(* PLC project CoDeSys External Library Template, WAGO e!COCKPIT e!COCKPIT, author 3S - Smart Software Solutions GmbH *)
(* stored: creationDateTime 2019-10-29T12:37:19.7040014, version 3.5.5.30, modificationDateTime 2019-10-29T12:36:39.3744516, organization 3S - Smart Software Solutions GmbH *)
(* Library project template with all possible element types, docu and a sample project structure *)

FUNCTION_BLOCK fbPPPSSilownikSABp
  VAR_INPUT
    sKomunikat : alSTRINGKomunikat;  (* komunikat z systemu zewnętrznego *)
    intTablicaKomunikatowRozmiar : INT;  (* rozmiar tablicy danych wysyłkowych *)
    intModbusOdczytZapisZadanieRozmiar : INT;  (* rozmiar tablicy danych modbusa *)
    xTablicaKomunikatowHold : BOOL;  (* wstrzymanie komunikacji mniej ważnych komunikatów *)
    sIdInstancji : STRING;  (* parametr ID rolety np NS02L*202IBM**** *)
    sIdAplikacji : STRING;  (* parametr ID aplikacji np SO*******ECL*000 *)
    sMnemonik : STRING;  (* mnemonik właściciela - BCB* *)
    sMACAdres : STRING;  (* MAC adres sterownika *)
    sDaneZapasowe : STRING;  (* 6 znaków zapasu *)
    tCzasOpoznieniaRestartu : TIME;  (* czas opóźnienia po którym zaczynają być raportowane wartości *)
    bAdres : BYTE;
    bKanalEnOcean : BYTE;
    sEnOceanID : STRING(10);
    rZadanePolozenieSilownika : REAL;
    tMinimalnyCzasRaportowania : TIME;
    tMaksymalnyCzasRaportowania : TIME;
    tCzasTimeoutEnOcean : TIME;
    xAutonomizacja : BOOL;
    xAutonomizacjaSztuczna : BOOL;
    xGlobalnaAutomatycznaKonfiguracja : BOOL;
    tCzestotliwoscAutomatycznejKonfiguracji : TIME;
    rTrybPracyAutonomizacja : REAL;  (* Domyślny tryb pracy *)
    rPozycjaSilownikaManAutonomizacja : REAL;  (* Domyślne położenie siłownika *)
    rFlagaSerwisowaAutonomizacja : REAL;  (* Domyślna flaga serwisowa *)
    tCzasSpadkuTemperatury : TIME;  (* Okres detekcji *)
    rDeltaSpadkuTemperatury : REAL;  (* Wartość o jaką musi spaść temp. w okresie intCzasSpadkuTemperatury, aby wyzwolić alarm *)
    rDeltaWzrostuTemperatury : REAL;  (* Wartość o jaką musi wzrosnąć temp. w okresie intCzasSpadkuTemperatury, aby odwołać alarm *)
    intTrybPracyHMI : INT := 1;  (* patrz enumPPPSZadajnikTrybPracy *)
    rZadanePolozenieSilownikaHMI : REAL;  (* Pozycja siłownika z nastawy na webvisu *)
    xPokazPanelHMI : BOOL := TRUE;  (* 0 - widoczny; 1 - niewidoczny *)
    xUsuwaniePotwierdzenieHMI : BOOL := FALSE;  (* wyświetlenie okienka potwierdzenia chęci usunięcia siłownika *)
    xUczenieWlaczHMI : BOOL := FALSE;  (* Włączenie flagi uczenia siłownika *)
    xUczenieWlaczone : BOOL;  (* Potwierdzenie włączenia uczenia *)
    xUsuwanieHMI : BOOL := FALSE;  (* Usuwanie EnOcean ID z kanału bramki *)
  END_VAR
  VAR_IN_OUT
    arModbusOdczytCykliczny : ARRAY[1..5000] OF typModbusOdczytCykliczny;
    arModbusStatusKomunikacji : ARRAY[1..256] OF INT;
    arModbusOdczytZapisZadanie : ARRAY[1..1000] OF typModbusOdczytZapisZadanie;
    intModbusOdczytZapisZadanieZnacznikZapisu : INT;
    arTablicaKomunikatow : alARRAYTablicaKomunikatow;
    intTablicaKomunikatowZnacznikZapisu : INT;
  END_VAR
  VAR_OUTPUT
    rDiagnostykaTemperaturaPomieszczenia : REAL;
    rDiagnostykaPozycjaSilownika : REAL;
    intDiagnostykaFlagaSerwisowa : INT;
    intDiagnostykaTrybPracy : INT;
    xDiagnostykaDetekcjaOtwarciaOkna : BOOL;
    sDiagnostykaEnOceanIDodczytany : STRING(10);
    xDiagnostykaPoprawneParowanie : BOOL;
    wDiagnostykaCzasOdOstatniegoKomunikatu : WORD;
  END_VAR
  VAR CONSTANT
    uintLiczbaRejestrowNaKanal : UINT := 20;
    uintPierwszyRejestr : UINT := 2000;
  END_VAR
  VAR
    wLearnEnOceanOdczytany : WORD;
    xLearnEnOceanOdczytany : BOOL;
    xLearnEnOceanWlacz : BOOL;
    xLearnEnOceanWylacz : BOOL;
    fbWysylanieLearn : TON;
    intTemp : INT := 0;
    xResetWysylanieLern : BOOL;
    xPoprawneParowanie : BOOL;
    uintORGModbusAdres : UINT;  (* definicja adresów rejestrów modbusowych *)
    uintFunctionModbusAdres : UINT;
    uintTypeModbusAdres : UINT;
    uintManufacturerModbusAdres : UINT;
    uintEnOceanIDHiModbusAdres : UINT;
    uintEnOceanIDLoModbusAdres : UINT;
    uintCzasOdOstatniegoKomunikatuModbusAdres : UINT;
    uintZadanaPozycjaSilownikaModbusAdres : UINT;
    uintFlagaSerwisowaModbusAdres : UINT;
    uintStatusUrzadzeniaModbusAdres : UINT;
    uintTemperaturaPomieszczeniaOdczytanaModbusAdres : UINT;
    uintNastawaPotencjometraModbusAdres : UINT;
    uintUczenieSilownikaAdres : UINT := 31;  (* uintLiczbaTelegramowModbusAdres : UINT; *)
    uintLearnModbusAdres : UINT;
    xPierwszySkan : BOOL := TRUE;  (* zmienne operacyjne *)
    intPetlaPierwszySkan : INT := 1;
    intRozkazTymczasowy : INT;
    rtrigPrzywrocDomyslne : R_TRIG;  (* Przywracanie domyślnych wartości nastaw *)
    rtrigZapisModbus : R_TRIG;  (* Triger zapisu danych po Modbusie *)
    fbTaktowanieZapisywaniaModbus : TON;  (* Cykliczne żądanie zapisu danych do urządzenia *)
    tonBrakKomunikacjiPLC : TON;  (* Kontrola komunikacji urządzenia *)
    xBrakKomunikacjiPLC : BOOL;
    xBrakKomunikacjiIZE : BOOL;
    fbWyslanieKonfiguracji : TON;  (* definicja zmiennych i FB do odczytu wartości z modbusa *)
    xPozwolenieNaAutomatycznaKonfiguracje : BOOL;
    xResetTimerautomatycznejKonfiguracji : BOOL;
    intBlokadaWykonywaniaRozkazow : INT;
    intBlokadaWykonywaniaRozkazowZaraportowana : INT;
    intTrybPracy : INT;  (* Tryb pracy regulatora. *)
    intTrybPracyPamiec : INT;
    intTrybPracyZaraportowana : INT;
    xTrybPracyZapisz : BOOL;  (* Trigger zapisu wartości w pamięci urządzenia. *)
    rTrybPracyZapis : REAL;  (* Wartość do zapisania w pamięci urządzenia. *)
    wFunctionEnOceanOdczytana : WORD;
    wTypeEnOceanOdczytana : WORD;
    wManufacturerEnOceanOdczytana : WORD;
    sEnOceanIDodczytany : STRING(10);
    wEnOceanIDHi : WORD;
    wEnOceanIDLo : WORD;
    wEnOceanIDHiZapis : WORD;
    wEnOceanIDLoZapis : WORD;
    wCzasOdOstatniegoKomunikatu : WORD;
    fbTimeoutEnOcean : TON;
    wStatusUrzadzenia : WORD;
    xBladBaterii : BOOL;
    fbBladBaterii : TON;
    xAlarmOgolny : BOOL;
    fbDecToBin : fbDecToBin;
    wLiczbaTelegramow : WORD;
    uintLiczbaTelegramow : UINT;
    wTemperaturaPomieszczeniaOdczytana : WORD;
    fbTemperaturaPomieszczenia : fbFiltrWartoscAnalogowa;
    rTemperaturaPomieszczenia : REAL := 273.15;
    rTemperaturaPomieszczeniaZaraportowana : REAL;
    rTemperaturaPomieszczeniaPamiec : REAL;  (* Temperatura zapamiętana w celu porównania z aktualną *)
    xBrakZmianyTemperatury : BOOL;  (* Flaga braku zmiany temperatury *)
    fbBrakZmianyTemperaturyTimer : TON;  (* Timer braku zmiany temperatury (24 godziny) *)
    xBladBrakZmianyTemperatury : BOOL;  (* Błąd braku zmiany temperatury *)
    wPozycjaSilownikaOdczytana : WORD;
    wPozycjaSilownikaZadanie : WORD;
    fbPozycjaSilownika : fbFiltrWartoscAnalogowa;
    rPozycjaSilownika : REAL;  (* Pozycja siłownika. *)
    rPozycjaSilownikaZaraportowana : REAL;
    rPozycjaSilownikaAuto : REAL;  (* Pozycja siłownika w trybie automatycznym. *)
    rPozycjaSilownikaAutoZaraportowana : REAL;
    rPozycjaSilownikaMan : REAL;  (* Pozycja siłownika w trybie manualnym *)
    rPozycjaSilownikaManZaraportowana : REAL;
    xPozycjaSilownikaManZapisz : BOOL;  (* Trigger zapisu wartości w pamięci urządzenia. *)
    rPozycjaSilownikaManZapis : REAL;  (* Wartość do zapisania w pamięci urządzenia. *)
    fbUtrzymaniaPolozeniaAutonomizacja : TON;
    xRestartTimeraUtrzymaniaPolozeniaAutonomizacja : BOOL;
    xWykonanoZapisPolozeniaSilownika : BOOL := FALSE;
    tCzasWyslaniaKomunikatuZapisuPozycjiSilownika : TIME;
    wFlagaSerwisowaOdczytana : WORD;
    wFlagaSerwisowaZadanie : WORD;
    intFlagaSerwisowa : INT;
    intFlagaSerwisowaZaraportowana : INT;
    xFlagaSerwisowaZapisz : BOOL;  (* Trigger zapisu wartości w pamięci urządzenia. *)
    rFlagaSerwisowaZapis : REAL;  (* Wartość do zapisania w pamięci urządzenia. *)
    xZmianaFlagiSerwisowejNaBrakDzialan : BOOL;
    xZmianaFlagiSerwisowejNaTrybLetni : BOOL;
    xZmianaFlagiSerwisowejNaZamkniecieZaworu : BOOL;
    xZmianaFlagiSerwisowejNaOtwarcieZaworu : BOOL;
    xZmianaFlagiSerwisowejNaPozycjaGorna : BOOL;
    xZmianaFlagiSerwisowejNaKalibracjeSilownika : BOOL;
    fbTimerZmianyFlagiSerwisowej : TON;
    xPoInicjalizacji : BOOL := FALSE;  (* inicjalizacja *)
    fbInicjalizacyjnyTimer : TON;
    sDane : alSTRINGKomunikat;
    sWyslanyKomunikat : alSTRINGKomunikat;
    sKomunikatPamiec : alSTRINGKomunikat;
    sWyslanyKomunikatDummy : alSTRINGKomunikat;
    intPetla : INT;
    arErrorStan : ARRAY[0..5] OF INT;  (* tablica przechowująca statusy alarmowe *)
    arErrorKlasa : ARRAY[0..5] OF INT;  (* tablica przechowująca klasy danych alarmów *)
    sTempWartoscAtrybutu : STRING;
    xRaport : BOOL;
    rNastawaPolozeniaSilownika : REAL;
    xAlarmOtwarciaOkna : BOOL;  (* Alarm detekcji gwałtownego spadku temperatury siłownika (otwarcia okna nad grzejnikiem) *)
    rTemperaturaPomieszczeniaHistoryczna : REAL;  (* Wartość temperatury zapisywana co intCzasSpadkuTemperatury w celu obliczenia różnicy *)
    fbDetekcjaOtwarciaOknaTimer : TON;  (* Timer detekcji otwarcia okna *)
    xDefrost : BOOL;  (* Defrost *)
    fbDefrostTimer : TON;
    rtrigDefrostTimer : R_TRIG;
    fbDefrostOdwolanie : TON;
    fnUczenieTimer : TON;  (* Timer uczenia *)
    fnWlaczenieUczenia : R_TRIG;  (* Włączenie uczenie na panelu HMI *)
    fnWylaczenieUczenia : F_TRIG;  (* Wyłączenie uczenia na panelu HMI *)
    fnUczenieZakonczone : F_TRIG;  (* Uczenie zostało zakończone *)
    xBrakKomunikacjiEnOcean : BOOL;  (* Brak komunikacji z urządzeniem po enOcean *)
    xAwariaUrzadzenia : BOOL;  (* Alarm ogólny *)
    rTempWartoscAtrybutu : REAL;
    intTempWartoscAtrybutu : INT;
    xDetekcjaOtwarciaOkna : BOOL;
  END_VAR

            (*			
Autor:					Paweł Kąkol, 2018-08-23-PK; Artur Wyszomirski; Jan Bartczak
Prawa majątkowe: 		Solwena Sp. z o.o., 
Aktualizacje:			
						2018-08-27-PK: dodanie algorytmu nadpisywania konfiguracji (uczenia) anteny
						2018-09-04-PK: dodanie rozkazu C, dodanie zapytań Q, dodanie raportowania M, dodanie alarmowania
						2018-09-10-PK: zmiana alarmowania braku komunikacji z Modbus RTU na alarmowanie timeout komunikacji EnOcean
						2018-09-12-PK: zaremowanie kodu uczącego bramkę, dodanie możliwości uczenia (LearnMode) ze zmiennej BOOL, sprawdzanie poprawności zainstalowania urządzenia (po EnOceanID)
						2018-09-25-AW: obsługa trybów manualnego i automatycznego
						2018-10-01-JB: dodanie ręcznej zmiany flagi serwisowej siłownika, zmiana sposobu zapisywania wartości wysterowania siłownika 
						2018-10-03-JB: poprawienie odczytywania kodów błędów
						2018-23-10-JB: przygotowanie atrybutów i alarmów do komunikacji z IZE
						2018-11-16-AW: inicjalizacja uczenia siłowników z programy
						2018-12-11-JB: zmiana sposobu działania alarmu z błędem baterii. Do momentu pierwszego odczytu wartości za pomocą ModbusRTU generowała się błędna informacja o błędzie baterii. 			
						2018-12-11-JB: skasowanie obsługi detekcji okna, ponieważ ten siłownik tego nie zawiera. 	
						2018-12-12-JB: napisanie od nowa obsługi ramek typu C i Q
						2019-01-04-AWy: detekcja otwarcia okna
						2019-01-28-JC: defrost
						2019-02-14-AWy: wysyłanie alarmu czujnika temperatury
						2019-02-27-JB: zmiana deadbandów w filtrach analogowych
						2019-03-20-AWy: uczenie siłownika z poziomu panelu HMI
						2019-03-21-AWy: usuwanie siłownika z poziomu panelu HMI
						2019-05-16-AWy: modyfikacja warunku na raportowanie. Dopisane: AND arModbusStatusKomunikacji[bAdres] = enumModbusStatus.KomunikacjaPrawidlowa AND xPoInicjalizacji 
						2019-05-20-AWy: - zmiana zachowania Defrostu. Po wykryciu spadku temperatury poniżej 8 stopni następuje przełączenie w tryb ręczny i odpalanie siłownika na 100%. 
										- alarm odwołany i powrót do normalnej pracy po osiągnięciu temperatury powyżej 10 stopni.
						2019-06-06-AWy: załadowanie domyślnych trybów pracy i nastaw po przejściu w tryb autonomizacji.
						2019-08-14-AWy: zmiana algorytmu defrostu ze względu na zmianę sposobu wybierania trybów pracy. Zmiana fbPrzywrocDomyslne z przerzutnika RS na R_TRIG.
						2019-09-17-AWy: usunięcie buga z defrostu.
						2019-09-23-AWy: modyfikacja generowania wartości zmiennej xBrakKomunikacjiPLC.
						2019-10-09-AWy: uzależnienie wystąpienia alarmu braku zmiany temperatury od stanu komunikacji.
						2019-10-18-AWy: dodanie atrybutu POZ.
						2019-10-22-AWy: - usunięcie uintLiczbaTelegramowModbusAdres z odczytu po Modbusie;
										- wydłużenie czasu fbTaktowanieZapisywaniaModbus oraz wprowadzenie trigera zapisu po Modbusie;
										- dodanie warunku poprawnej komunikacji przy generowaniu defrostu.
						2019-10-24-AWy: zmiana deadbandu fbPozycjaSilownika
												
Opis:					fb służy do komunikacji po Modbus RTU za pośrednictwem bramek (STC65-RS485) EnOcean z siłownikami HRU0 (SAB+) na budynkach PPP Sopot (ENGIE) 
*)

// Inicjalizacja sterownika
fbInicjalizacyjnyTimer(IN := NOT xPoInicjalizacji , PT := tCzasOpoznieniaRestartu);
IF fbInicjalizacyjnyTimer.Q THEN
	rTemperaturaPomieszczeniaZaraportowana := rTemperaturaPomieszczenia;
	rPozycjaSilownikaZaraportowana := rPozycjaSilownika;
	rPozycjaSilownikaAutoZaraportowana := rPozycjaSilownikaAuto;
	rPozycjaSilownikaManZaraportowana := rPozycjaSilownikaMan;
	intFlagaSerwisowaZaraportowana := intFlagaSerwisowa;
	xPoInicjalizacji := TRUE;
END_IF

// Włącz autonomizację jeśli sterownik jest w stanie inicjalizacji lub nastąpiło wymuszenie autonomizacji
IF NOT xPoInicjalizacji OR xAutonomizacjaSztuczna = TRUE THEN
	xAutonomizacja := TRUE;
END_IF 

// Kontrola komunikacji
tonBrakKomunikacjiPLC(IN := (wCzasOdOstatniegoKomunikatu > 180 OR arModbusStatusKomunikacji[bAdres] <> enumModbusStatus.KomunikacjaPrawidlowa), PT := T#180S);
IF tonBrakKomunikacjiPLC.Q THEN
	xBrakKomunikacjiPLC := TRUE;
ELSE
	xBrakKomunikacjiPLC := FALSE;
END_IF

IF xAutonomizacja THEN
	xBrakKomunikacjiIZE := TRUE;
ELSE
	xBrakKomunikacjiIZE := FALSE;
END_IF

// Deklaracja rejestrów Modbusa
IF xPierwszySkan THEN
	xPierwszySkan := FALSE;
	WHILE arModbusOdczytCykliczny[intPetlaPierwszySkan].bAdresUrzadzenia <> 0 DO
		intPetlaPierwszySkan := intPetlaPierwszySkan + 1;
	END_WHILE
	
	//wyznaczenie adresów rejestrów modbusowych
	uintORGModbusAdres := uintPierwszyRejestr + (uintLiczbaRejestrowNaKanal * (BYTE_TO_UINT(bKanalEnOcean) - 1));
	uintFunctionModbusAdres := uintORGModbusAdres + 1;
	uintTypeModbusAdres := uintORGModbusAdres + 2;
	uintManufacturerModbusAdres := uintORGModbusAdres + 3;
	uintEnOceanIDHiModbusAdres := uintORGModbusAdres + 4;
	uintEnOceanIDLoModbusAdres := uintORGModbusAdres + 5;
	uintCzasOdOstatniegoKomunikatuModbusAdres := uintORGModbusAdres + 6;
	uintZadanaPozycjaSilownikaModbusAdres := uintORGModbusAdres + 7;
	uintFlagaSerwisowaModbusAdres := uintORGModbusAdres + 8;
	uintStatusUrzadzeniaModbusAdres := uintORGModbusAdres + 9;
	uintTemperaturaPomieszczeniaOdczytanaModbusAdres := uintORGModbusAdres + 10;
	//uintLiczbaTelegramowModbusAdres := uintORGModbusAdres + 19;
	
	uintLearnModbusAdres := 31 + BYTE_TO_UINT(bKanalEnOcean);
	
//deklaracja rejestrow do odczytu
	//coil
	arModbusOdczytCykliczny[intPetlaPierwszySkan].bAdresUrzadzenia := bAdres;
	arModbusOdczytCykliczny[intPetlaPierwszySkan].bFunkcja := TO_BYTE(enumModbusKodyFunkcji.OdczytWyjscBitowych);
	arModbusOdczytCykliczny[intPetlaPierwszySkan].uiAdresRejestru := uintLearnModbusAdres;
	arModbusOdczytCykliczny[intPetlaPierwszySkan].ltCzestotliwosc := LTIME#1S;
	arModbusOdczytCykliczny[intPetlaPierwszySkan].pZmiennaReferencyjna := ADR(wLearnEnOceanOdczytany);
	intPetlaPierwszySkan := intPetlaPierwszySkan + 1;
	//rejestry
	arModbusOdczytCykliczny[intPetlaPierwszySkan].bAdresUrzadzenia := bAdres;
	arModbusOdczytCykliczny[intPetlaPierwszySkan].bFunkcja := TO_BYTE(enumModbusKodyFunkcji.OdczytNRejestrow);
	arModbusOdczytCykliczny[intPetlaPierwszySkan].uiAdresRejestru := uintFunctionModbusAdres;
	arModbusOdczytCykliczny[intPetlaPierwszySkan].ltCzestotliwosc := TIME_TO_LTIME(tMinimalnyCzasRaportowania);
	arModbusOdczytCykliczny[intPetlaPierwszySkan].pZmiennaReferencyjna := ADR(wFunctionEnOceanOdczytana);
	intPetlaPierwszySkan := intPetlaPierwszySkan + 1;
	
	arModbusOdczytCykliczny[intPetlaPierwszySkan].bAdresUrzadzenia := bAdres;
	arModbusOdczytCykliczny[intPetlaPierwszySkan].bFunkcja := TO_BYTE(enumModbusKodyFunkcji.OdczytNRejestrow);
	arModbusOdczytCykliczny[intPetlaPierwszySkan].uiAdresRejestru := uintTypeModbusAdres;
	arModbusOdczytCykliczny[intPetlaPierwszySkan].ltCzestotliwosc := TIME_TO_LTIME(tMinimalnyCzasRaportowania);
	arModbusOdczytCykliczny[intPetlaPierwszySkan].pZmiennaReferencyjna := ADR(wTypeEnOceanOdczytana);
	intPetlaPierwszySkan := intPetlaPierwszySkan + 1;
	
	arModbusOdczytCykliczny[intPetlaPierwszySkan].bAdresUrzadzenia := bAdres;
	arModbusOdczytCykliczny[intPetlaPierwszySkan].bFunkcja := TO_BYTE(enumModbusKodyFunkcji.OdczytNRejestrow);
	arModbusOdczytCykliczny[intPetlaPierwszySkan].uiAdresRejestru := uintManufacturerModbusAdres;
	arModbusOdczytCykliczny[intPetlaPierwszySkan].ltCzestotliwosc := TIME_TO_LTIME(tMinimalnyCzasRaportowania);
	arModbusOdczytCykliczny[intPetlaPierwszySkan].pZmiennaReferencyjna := ADR(wManufacturerEnOceanOdczytana);
	intPetlaPierwszySkan := intPetlaPierwszySkan + 1;
	
	arModbusOdczytCykliczny[intPetlaPierwszySkan].bAdresUrzadzenia := bAdres;
	arModbusOdczytCykliczny[intPetlaPierwszySkan].bFunkcja := TO_BYTE(enumModbusKodyFunkcji.OdczytNRejestrow);
	arModbusOdczytCykliczny[intPetlaPierwszySkan].uiAdresRejestru := uintEnOceanIDHiModbusAdres;
	arModbusOdczytCykliczny[intPetlaPierwszySkan].ltCzestotliwosc := TIME_TO_LTIME(tMinimalnyCzasRaportowania);
	arModbusOdczytCykliczny[intPetlaPierwszySkan].pZmiennaReferencyjna := ADR(wEnOceanIDHi);
	intPetlaPierwszySkan := intPetlaPierwszySkan + 1;
	
	arModbusOdczytCykliczny[intPetlaPierwszySkan].bAdresUrzadzenia := bAdres;
	arModbusOdczytCykliczny[intPetlaPierwszySkan].bFunkcja := TO_BYTE(enumModbusKodyFunkcji.OdczytNRejestrow);
	arModbusOdczytCykliczny[intPetlaPierwszySkan].uiAdresRejestru := uintEnOceanIDLoModbusAdres;
	arModbusOdczytCykliczny[intPetlaPierwszySkan].ltCzestotliwosc := TIME_TO_LTIME(tMinimalnyCzasRaportowania);
	arModbusOdczytCykliczny[intPetlaPierwszySkan].pZmiennaReferencyjna := ADR(wEnOceanIDLo);
	intPetlaPierwszySkan := intPetlaPierwszySkan + 1;
	
	arModbusOdczytCykliczny[intPetlaPierwszySkan].bAdresUrzadzenia := bAdres;
	arModbusOdczytCykliczny[intPetlaPierwszySkan].bFunkcja := TO_BYTE(enumModbusKodyFunkcji.OdczytNRejestrow);
	arModbusOdczytCykliczny[intPetlaPierwszySkan].uiAdresRejestru := uintCzasOdOstatniegoKomunikatuModbusAdres;
	arModbusOdczytCykliczny[intPetlaPierwszySkan].ltCzestotliwosc := TIME_TO_LTIME(tMinimalnyCzasRaportowania);
	arModbusOdczytCykliczny[intPetlaPierwszySkan].pZmiennaReferencyjna := ADR(wCzasOdOstatniegoKomunikatu);
	intPetlaPierwszySkan := intPetlaPierwszySkan + 1;
	
	arModbusOdczytCykliczny[intPetlaPierwszySkan].bAdresUrzadzenia := bAdres;
	arModbusOdczytCykliczny[intPetlaPierwszySkan].bFunkcja := TO_BYTE(enumModbusKodyFunkcji.OdczytNRejestrow);
	arModbusOdczytCykliczny[intPetlaPierwszySkan].uiAdresRejestru := uintZadanaPozycjaSilownikaModbusAdres;
	arModbusOdczytCykliczny[intPetlaPierwszySkan].ltCzestotliwosc := TIME_TO_LTIME(tMinimalnyCzasRaportowania);
	arModbusOdczytCykliczny[intPetlaPierwszySkan].pZmiennaReferencyjna := ADR(wPozycjaSilownikaOdczytana);
	intPetlaPierwszySkan := intPetlaPierwszySkan + 1;	
	
	arModbusOdczytCykliczny[intPetlaPierwszySkan].bAdresUrzadzenia := bAdres;
	arModbusOdczytCykliczny[intPetlaPierwszySkan].bFunkcja := TO_BYTE(enumModbusKodyFunkcji.OdczytNRejestrow);
	arModbusOdczytCykliczny[intPetlaPierwszySkan].uiAdresRejestru := uintFlagaSerwisowaModbusAdres;
	arModbusOdczytCykliczny[intPetlaPierwszySkan].ltCzestotliwosc := TIME_TO_LTIME(tMinimalnyCzasRaportowania);
	arModbusOdczytCykliczny[intPetlaPierwszySkan].pZmiennaReferencyjna := ADR(wFlagaSerwisowaOdczytana);
	intPetlaPierwszySkan := intPetlaPierwszySkan + 1;
	
	arModbusOdczytCykliczny[intPetlaPierwszySkan].bAdresUrzadzenia := bAdres;
	arModbusOdczytCykliczny[intPetlaPierwszySkan].bFunkcja := TO_BYTE(enumModbusKodyFunkcji.OdczytNRejestrow);
	arModbusOdczytCykliczny[intPetlaPierwszySkan].uiAdresRejestru := uintStatusUrzadzeniaModbusAdres;
	arModbusOdczytCykliczny[intPetlaPierwszySkan].ltCzestotliwosc := TIME_TO_LTIME(tMinimalnyCzasRaportowania);
	arModbusOdczytCykliczny[intPetlaPierwszySkan].pZmiennaReferencyjna := ADR(wStatusUrzadzenia);
	intPetlaPierwszySkan := intPetlaPierwszySkan + 1;
	
	arModbusOdczytCykliczny[intPetlaPierwszySkan].bAdresUrzadzenia := bAdres;
	arModbusOdczytCykliczny[intPetlaPierwszySkan].bFunkcja := TO_BYTE(enumModbusKodyFunkcji.OdczytNRejestrow);
	arModbusOdczytCykliczny[intPetlaPierwszySkan].uiAdresRejestru := uintTemperaturaPomieszczeniaOdczytanaModbusAdres;
	arModbusOdczytCykliczny[intPetlaPierwszySkan].ltCzestotliwosc := TIME_TO_LTIME(tMinimalnyCzasRaportowania);
	arModbusOdczytCykliczny[intPetlaPierwszySkan].pZmiennaReferencyjna := ADR(wTemperaturaPomieszczeniaOdczytana);
	intPetlaPierwszySkan := intPetlaPierwszySkan + 1;
(*	
	arModbusOdczytCykliczny[intPetlaPierwszySkan].bAdresUrzadzenia := bAdres;
	arModbusOdczytCykliczny[intPetlaPierwszySkan].bFunkcja := TO_BYTE(enumModbusKodyFunkcji.OdczytNRejestrow);
	arModbusOdczytCykliczny[intPetlaPierwszySkan].uiAdresRejestru := uintLiczbaTelegramowModbusAdres;
	arModbusOdczytCykliczny[intPetlaPierwszySkan].ltCzestotliwosc := TIME_TO_LTIME(tMinimalnyCzasRaportowania);
	arModbusOdczytCykliczny[intPetlaPierwszySkan].pZmiennaReferencyjna := ADR(wLiczbaTelegramow);
	intPetlaPierwszySkan := intPetlaPierwszySkan + 1;
*)			
	arModbusOdczytCykliczny[intPetlaPierwszySkan].bAdresUrzadzenia := bAdres;
	arModbusOdczytCykliczny[intPetlaPierwszySkan].bFunkcja := TO_BYTE(enumModbusKodyFunkcji.OdczytWyjscBitowych);
	arModbusOdczytCykliczny[intPetlaPierwszySkan].uiAdresRejestru := uintUczenieSilownikaAdres + BYTE_TO_UINT(bKanalEnOcean);
	arModbusOdczytCykliczny[intPetlaPierwszySkan].ltCzestotliwosc := TIME_TO_LTIME(tMinimalnyCzasRaportowania);
	arModbusOdczytCykliczny[intPetlaPierwszySkan].pZmiennaReferencyjna := ADR(xUczenieWlaczone);
	intPetlaPierwszySkan := intPetlaPierwszySkan + 1;
END_IF

//obsluga komunikatu przychodzacego z IZE

IF 	sKomunikat <> sKomunikatPamiec AND xPoInicjalizacji THEN
	sKomunikatPamiec := sKomunikat;
	IF fnIDOdbiorcyMatch(sKomunikat , sIdInstancji) THEN
		sDane := '';
		//rozkaz typu C
		IF fnKomunikatTyp(sKomunikat) = 'C' AND NOT xAutonomizacja THEN
		//blokada
			IF fnKomunikatDaneSzukajWartosci(sKomunikat,'BLOK=') = '0' THEN
				IF intBlokadaWykonywaniaRozkazow = 1 THEN
					intBlokadaWykonywaniaRozkazow := 0;
					xRaport := TRUE;
					ELSE	
					IF sDane <> '' THEN
					sDane := CONCAT(sDane , ';');
					END_IF
					sDane := CONCAT(sDane , 'BLOK=0');
				END_IF
			END_IF
			IF fnKomunikatDaneSzukajWartosci(sKomunikat,'BLOK=') = '1' THEN
				IF intBlokadaWykonywaniaRozkazow = 0 THEN
					intBlokadaWykonywaniaRozkazow := 1;
					xRaport := TRUE;
					ELSE
					IF sDane <> '' THEN
					sDane := CONCAT(sDane , ';');
					END_IF					
					sDane := CONCAT(sDane , 'BLOK=1');
				END_IF
			END_IF
			
			IF intBlokadaWykonywaniaRozkazow = 0 THEN
				// Tryby pracy 
				fnKomunikatDaneZnajdzPorownajZapisz(sKomunikat := sKomunikat,
					sAtrybut := 'TRYB=',
					rAtrybutWartosc := rTrybPracyZapis,
					sDane := sDane,
					xAtrybutZapisz => xTrybPracyZapisz);		
				// Pozycja siłownika w trybie manualnym
				fnKomunikatDaneZnajdzPorownajZapisz(sKomunikat := sKomunikat,
					sAtrybut := 'POZMAN=',
					rAtrybutWartosc := rPozycjaSilownikaManZapis,
					sDane := sDane,
					xAtrybutZapisz => xPozycjaSilownikaManZapisz);
				// Flaga serwisowa
				fnKomunikatDaneZnajdzPorownajZapisz(sKomunikat := sKomunikat,
					sAtrybut := 'SERWIS=',
					rAtrybutWartosc := rFlagaSerwisowaZapis,
					sDane := sDane,
					xAtrybutZapisz => xFlagaSerwisowaZapisz);	
			END_IF	
		END_IF		

		//zapytanie typu Q
		IF fnKomunikatTyp(sKomunikat) = 'Q' AND arModbusStatusKomunikacji[bAdres] = enumModbusStatus.KomunikacjaPrawidlowa THEN
			IF fnKomunikatDaneSzukajWartosci(sKomunikat , 'BLOK=') = '?' OR fnKomunikatDaneSzukajWartosci(sKomunikat , 'ALL=') = '?' THEN
				fnKomunikatDaneDodaj(sDane := sDane , sAtrybut := 'BLOK=' , sWartosc := INT_TO_STRING(intBlokadaWykonywaniaRozkazow));	
			END_IF
			IF fnKomunikatDaneSzukajWartosci(sKomunikat , 'TRYB=') = '?' OR fnKomunikatDaneSzukajWartosci(sKomunikat , 'ALL=') = '?' THEN
				fnKomunikatDaneDodaj(sDane := sDane , sAtrybut := 'TRYB=' , sWartosc := INT_TO_STRING(intTrybPracy));	
			END_IF
			IF fnKomunikatDaneSzukajWartosci(sKomunikat , 'TEMP=') = '?' OR fnKomunikatDaneSzukajWartosci(sKomunikat , 'ALL=') = '?' THEN
				fnKomunikatDaneDodaj(sDane := sDane , sAtrybut := 'TEMP=' , sWartosc := REAL_TO_STRING(rTemperaturaPomieszczenia));	
			END_IF
			IF fnKomunikatDaneSzukajWartosci(sKomunikat , 'POZ=') = '?' OR fnKomunikatDaneSzukajWartosci(sKomunikat , 'ALL=') = '?' THEN
				fnKomunikatDaneDodaj(sDane := sDane , sAtrybut := 'POZ=' , sWartosc := REAL_TO_STRING(rPozycjaSilownika));	
			END_IF
			IF fnKomunikatDaneSzukajWartosci(sKomunikat , 'POZAUTO=') = '?' OR fnKomunikatDaneSzukajWartosci(sKomunikat , 'ALL=') = '?' THEN
				fnKomunikatDaneDodaj(sDane := sDane , sAtrybut := 'POZAUTO=' , sWartosc := REAL_TO_STRING(rPozycjaSilownikaAuto));	
			END_IF
			IF fnKomunikatDaneSzukajWartosci(sKomunikat , 'POZMAN=') = '?' OR fnKomunikatDaneSzukajWartosci(sKomunikat , 'ALL=') = '?' THEN
				fnKomunikatDaneDodaj(sDane := sDane , sAtrybut := 'POZMAN=' , sWartosc := REAL_TO_STRING(rPozycjaSilownikaMan / 100));	
			END_IF
			IF fnKomunikatDaneSzukajWartosci(sKomunikat , 'SERWIS=') = '?' OR fnKomunikatDaneSzukajWartosci(sKomunikat , 'ALL=') = '?' THEN
				fnKomunikatDaneDodaj(sDane := sDane , sAtrybut := 'SERWIS=' , sWartosc := INT_TO_STRING(intFlagaSerwisowa));	
			END_IF
			//pytanie o stany alarmów
			IF fnKomunikatDaneSzukajWartosci(sKomunikat , 'ALARM=') = '?' OR fnKomunikatDaneSzukajWartosci(sKomunikat , 'ALL=') = '?' THEN
				FOR intPetla := 1 TO 5 BY 1 DO
					//raportowanie typu E (stanów alarmów) na zapytanie typu Q
					IF arErrorStan[intPetla] <> enumAlarmWartosc.StanNieznany THEN
						fnZapiszKomunikat(	sCalyKomunikat := '' ,
											sTypKomunikatu := 'E' ,
											sMnemonik := sMnemonik ,
											sMACAdres := sMACAdres ,
											sIDNadawcy := sIdInstancji ,
											sIDOdbiorcy := sIdAplikacji ,
											sDaneZapasowe := sDaneZapasowe ,
											sDane := fnKomunikatDaneErrorRetry(xAktywny := arErrorStan[intPetla] = enumAlarmWartosc.StanAlarmowy , intKlasa := arErrorKlasa[intPetla] , intNumer := intPetla),
											arTablicaKomunikatow := arTablicaKomunikatow ,
											intTablicaKomunikatowZnacznikZapisu := intTablicaKomunikatowZnacznikZapisu ,
											intTablicaKomunikatowRozmiar := intTablicaKomunikatowRozmiar ,
											sWyslanyKomunikat := sWyslanyKomunikatDummy);
					END_IF
				END_FOR
			END_IF
		END_IF
		//raportowanie typu A
		IF sDane <> '' THEN
			fnZapiszKomunikat(	sCalyKomunikat := '' ,
								sTypKomunikatu := 'A' ,
								sMnemonik := sMnemonik ,
								sMACAdres := sMACAdres ,
								sIDNadawcy := sIdInstancji ,
								sIDOdbiorcy := sIdAplikacji ,
								sDaneZapasowe := sDaneZapasowe ,
								sDane := sDane ,
								arTablicaKomunikatow := arTablicaKomunikatow ,
								intTablicaKomunikatowZnacznikZapisu := intTablicaKomunikatowZnacznikZapisu ,
								intTablicaKomunikatowRozmiar := intTablicaKomunikatowRozmiar ,
								sWyslanyKomunikat := sWyslanyKomunikatDummy);
		END_IF
	END_IF
END_IF

// Przywrócenie wartości domyślnych nastaw krzywej grzewczej i trybów pracy w przypadku restartu sterownika lub przejścia w stan autonomizacji (brak komunikacji z IZE)
rtrigPrzywrocDomyslne(CLK := xAutonomizacja);
IF rtrigPrzywrocDomyslne.Q THEN	
	IF intTrybPracy <> REAL_TO_INT(rTrybPracyAutonomizacja) THEN
		rTrybPracyZapis := rTrybPracyAutonomizacja;
		xTrybPracyZapisz := TRUE;
	END_IF
	IF rPozycjaSilownikaMan <> rPozycjaSilownikaManAutonomizacja THEN
		rPozycjaSilownikaManZapis := rPozycjaSilownikaManAutonomizacja / 100;
		xPozycjaSilownikaManZapisz := TRUE;
	END_IF
	IF intFlagaSerwisowa <> REAL_TO_INT(rFlagaSerwisowaAutonomizacja) THEN
		rFlagaSerwisowaZapis :=  rFlagaSerwisowaAutonomizacja;
		xFlagaSerwisowaZapisz := TRUE;
	END_IF
END_IF	

// Zapisanie nastaw domyślnych lub otrzymanych w ramce C
IF xTrybPracyZapisz THEN
	intTrybPracy := REAL_TO_INT(rTrybPracyZapis);
	intTrybPracyHMI := REAL_TO_INT(rTrybPracyZapis);
	xTrybPracyZapisz := FALSE;
END_IF	
IF xPozycjaSilownikaManZapisz THEN
	rPozycjaSilownikaMan := rPozycjaSilownikaManZapis * 100;
	xPozycjaSilownikaManZapisz := FALSE;
END_IF	

// Trigger zapisu po Modbusie
rtrigZapisModbus (CLK := xFlagaSerwisowaZapisz);

// Taktowanie zapisywania po Modbusie
fbTaktowanieZapisywaniaModbus(IN := NOT fbTaktowanieZapisywaniaModbus.Q, PT := T#180S);
				
// Zapisywanie trybu pracy do pamięci urządzenia
IF xFlagaSerwisowaZapisz AND (fbTaktowanieZapisywaniaModbus.Q OR rtrigZapisModbus.Q) THEN
	fnModbusZapisRejestru(	bAdresUrzadzenia := bAdres,
							bFunkcja := INT_TO_BYTE(enumModbusKodyFunkcji.ZapisRejestru),
							uiAdresRejestru := uintFlagaSerwisowaModbusAdres,
							pZmiennaReferencyjna := 0,
							wWartoscDoZapisania := REAL_TO_WORD(rFlagaSerwisowaZapis),
							intModbusOdczytZapisZadanieRozmiar := intModbusOdczytZapisZadanieRozmiar,
							arModbusOdczytZapisZadanie := arModbusOdczytZapisZadanie,
							intModbusOdczytZapisZadanieZnacznikZapisu := intModbusOdczytZapisZadanieZnacznikZapisu);
	IF intFlagaSerwisowa = REAL_TO_INT(rFlagaSerwisowaZapis) THEN					
		xFlagaSerwisowaZapisz := FALSE;
	END_IF
END_IF

//Auto konfiguracja anteny - sprawdzenie czy EnOcean ID wpisany w EiG jest zgodny z tym odczytanym z kanalu bramki
sEnOceanIDodczytany := CONCAT(CONCAT(fnKonwersjaDEC_BYTE_TO_HEX_STRING(INT_TO_BYTE(WORD_TO_INT(wEnOceanIDHi / 256))), fnKonwersjaDEC_BYTE_TO_HEX_STRING(WORD_TO_BYTE(wEnOceanIDHi))), CONCAT(fnKonwersjaDEC_BYTE_TO_HEX_STRING(INT_TO_BYTE(WORD_TO_INT(wEnOceanIDLo / 256))), fnKonwersjaDEC_BYTE_TO_HEX_STRING(WORD_TO_BYTE(wEnOceanIDLo))));
IF sEnOceanIDodczytany = sEnOceanID THEN
	xPoprawneParowanie := TRUE;
ELSE
	xPoprawneParowanie := FALSE;
END_IF

//sprawdzanie Timeout komunikacji
fbTimeoutEnOcean(IN := ((wCzasOdOstatniegoKomunikatu > 180 OR wCzasOdOstatniegoKomunikatu = 0) AND arModbusStatusKomunikacji[bAdres] = enumModbusStatus.KomunikacjaPrawidlowa) , PT := tCzasTimeoutEnOcean);

// dokonywanie obliczeń
fbTemperaturaPomieszczenia(	rWartoscWejsciowa := WORD_TO_REAL(wTemperaturaPomieszczeniaOdczytana),
							rWartoscWejsciowaZaraportowana := rTemperaturaPomieszczeniaZaraportowana,
							rDeadband := 0.1,
							tCzasMinimalny := tMinimalnyCzasRaportowania,
							tCzasMaksymalny := tMaksymalnyCzasRaportowania,
							rWynikMnoznik := 0.1,
							rWynikOffset := 273.15,
							rWartoscWyjsciowa => rTemperaturaPomieszczenia);
							
fbPozycjaSilownika(			rWartoscWejsciowa := WORD_TO_REAL(wPozycjaSilownikaOdczytana),
							rWartoscWejsciowaZaraportowana := rPozycjaSilownikaZaraportowana,
							rDeadband := 0.1,
							tCzasMinimalny := tMinimalnyCzasRaportowania,
							tCzasMaksymalny := tMaksymalnyCzasRaportowania,
							rWynikMnoznik := 0.01,
							rWynikOffset := 0.0,
							rWartoscWyjsciowa => rPozycjaSilownika);
							
CASE WORD_TO_INT(wFlagaSerwisowaOdczytana) OF
	0 : intFlagaSerwisowa := enumPPPSSilownikSABpServiceFlag.BrakDzialan;
	9 : intFlagaSerwisowa := enumPPPSSilownikSABpServiceFlag.TrybLetni;
	17 : intFlagaSerwisowa := enumPPPSSilownikSABpServiceFlag.ZamkniecieZaworu;
	33 : intFlagaSerwisowa := enumPPPSSilownikSABpServiceFlag.OtwarcieZaworu;
	65 : intFlagaSerwisowa := enumPPPSSilownikSABpServiceFlag.PozycjaGorna;
	129 : intFlagaSerwisowa := enumPPPSSilownikSABpServiceFlag.KalibracjaSilownika;
END_CASE
	
fbDecToBin(	wWordWejsciowy := wStatusUrzadzenia, 
			intIloscBitow := 8);
												
xAlarmOgolny := BYTE_TO_BOOL(fbDecToBin.arBity[0]);

// Defrost silownika. 
// Po spadku temperatury siłownika poniżej 8 stopni siłownik jest ustawiany w pozycję pełnego otwarcia (w trybie manualnym). Po wzroście temperatury powyżej 10 stopni siłownik powraca do trybu automatycznego.
fbDefrostTimer(IN := (rTemperaturaPomieszczenia < 281.15) AND (arModbusStatusKomunikacji[bAdres] = enumModbusStatus.KomunikacjaPrawidlowa), PT := T#5M);	// Temperatura poniżej 8 stopni C przez okres 5 minut
rtrigDefrostTimer(CLK := fbDefrostTimer.Q);
IF rtrigDefrostTimer.Q THEN
	intTrybPracyPamiec := intTrybPracy;	
END_IF

IF fbDefrostTimer.Q THEN	// Ustaw tryb pracy na manualny i otwórz zawór na 100%. Uruchom alarm
	rTrybPracyZapis := enumPPPSSilownikTrybPracy.Manualny;
	xTrybPracyZapisz := TRUE;
	rPozycjaSilownikaManZapis := 1;
	xPozycjaSilownikaManZapisz := TRUE;
	rZadanePolozenieSilownikaHMI := 100;
	xDefrost := TRUE;	
END_IF

fbDefrostOdwolanie(IN := ((rTemperaturaPomieszczenia > 283.15) AND xDefrost), PT := T#5M);	// Temperatura powyżej 10 stopni i uruchomiony Defrost przez okres 5 minut
IF fbDefrostOdwolanie.Q THEN	// Ustawa tryb pracy na automatyczny i odwołaj alarm
	rTrybPracyZapis := intTrybPracyPamiec;
	xTrybPracyZapisz := TRUE;
	xDefrost := FALSE;
END_IF
//
											
// Tryby pracy 
IF xAutonomizacja THEN	
	IF intTrybPracyHMI = enumPPPSSilownikTrybPracy.Manualny THEN								// tryb ręczny na HMI
		intTrybPracy := enumPPPSSilownikTrybPracy.Manualny;	
		rNastawaPolozeniaSilownika := rZadanePolozenieSilownikaHMI;
		rPozycjaSilownikaMan := rNastawaPolozeniaSilownika;
	ELSE																						// tryb automatyczny HMI
		intTrybPracy := enumPPPSSilownikTrybPracy.Automatyczny;	
		rNastawaPolozeniaSilownika := rZadanePolozenieSilownika;
		rZadanePolozenieSilownikaHMI := rZadanePolozenieSilownika;	
		rPozycjaSilownikaAuto := rPozycjaSilownika;											
	END_IF
ELSE
	rZadanePolozenieSilownikaHMI := rNastawaPolozeniaSilownika;
	IF intTrybPracy = enumPPPSSilownikTrybPracy.Manualny THEN
		rNastawaPolozeniaSilownika := rPozycjaSilownikaMan;
		intTrybPracyHMI := enumPPPSZadajnikTrybPracy.Manualny;
	ELSE
		rNastawaPolozeniaSilownika := rZadanePolozenieSilownika;
		intTrybPracyHMI := enumPPPSZadajnikTrybPracy.Automatyczny;
		rPozycjaSilownikaAuto := rPozycjaSilownika;		
	END_IF
END_IF
		
//utrzymanie położenia
fbUtrzymaniaPolozeniaAutonomizacja(IN := xRestartTimeraUtrzymaniaPolozeniaAutonomizacja = TRUE, PT := tCzasWyslaniaKomunikatuZapisuPozycjiSilownika);

IF (INT_TO_WORD(REAL_TO_INT(rNastawaPolozeniaSilownika)) <> wPozycjaSilownikaOdczytana) THEN
		xRestartTimeraUtrzymaniaPolozeniaAutonomizacja := TRUE;
		IF xWykonanoZapisPolozeniaSilownika = FALSE THEN
			tCzasWyslaniaKomunikatuZapisuPozycjiSilownika := T#5s;	
		END_IF	
ELSE
	xRestartTimeraUtrzymaniaPolozeniaAutonomizacja := FALSE;	
	xWykonanoZapisPolozeniaSilownika := FALSE;
END_IF

IF fbUtrzymaniaPolozeniaAutonomizacja.Q AND arModbusStatusKomunikacji[bAdres] = enumModbusStatus.KomunikacjaPrawidlowa THEN
	fnModbusZapisRejestru(	bAdresUrzadzenia := bAdres,
							bFunkcja := INT_TO_BYTE(enumModbusKodyFunkcji.ZapisRejestru),
							uiAdresRejestru := uintZadanaPozycjaSilownikaModbusAdres,
							pZmiennaReferencyjna := 0,
							wWartoscDoZapisania := (INT_TO_WORD(REAL_TO_INT(rNastawaPolozeniaSilownika))),
							intModbusOdczytZapisZadanieRozmiar := intModbusOdczytZapisZadanieRozmiar,
							arModbusOdczytZapisZadanie := arModbusOdczytZapisZadanie,
							intModbusOdczytZapisZadanieZnacznikZapisu := intModbusOdczytZapisZadanieZnacznikZapisu);
	xRestartTimeraUtrzymaniaPolozeniaAutonomizacja := FALSE;
	tCzasWyslaniaKomunikatuZapisuPozycjiSilownika := T#45s;
	xWykonanoZapisPolozeniaSilownika := TRUE;
END_IF

// Uczenie siłownika do bramki
fnWlaczenieUczenia(CLK := xUczenieWlaczHMI);
fnWylaczenieUczenia(CLK := xUczenieWlaczHMI);
fnUczenieZakonczone(CLK := xUczenieWlaczone);

IF fnUczenieZakonczone.Q OR fnUczenieTimer.Q THEN																		// Jeśli FALSE na coilu uczenia opuść toggla na HMI
	xUczenieWlaczHMI := FALSE;		
END_IF

IF fnWlaczenieUczenia.Q THEN						
	fnModbusZapisRejestru(	bAdresUrzadzenia := bAdres,																	// Wystawienie TRUE na coilu uczenia (patrz dok. STC65 rozdział 2.5.2)
							bFunkcja := INT_TO_BYTE(enumModbusKodyFunkcji.ZapisBitu),
							uiAdresRejestru := 31 + BYTE_TO_UINT(bKanalEnOcean),
							pZmiennaReferencyjna := 0,
							wWartoscDoZapisania := (BOOL_TO_WORD(TRUE)),
							intModbusOdczytZapisZadanieRozmiar := intModbusOdczytZapisZadanieRozmiar,
							arModbusOdczytZapisZadanie := arModbusOdczytZapisZadanie,
							intModbusOdczytZapisZadanieZnacznikZapisu := intModbusOdczytZapisZadanieZnacznikZapisu);	
END_IF

fnUczenieTimer(IN := xUczenieWlaczone, PT := T#1M);																		// Czas na uczenie - 1 minuta 

IF fnWylaczenieUczenia.Q THEN
	fnModbusZapisRejestru(	bAdresUrzadzenia := bAdres,																	// Wystawienie FALSE na coilu uczenia (patrz dok. STC65 rozdział 2.5.2)
							bFunkcja := INT_TO_BYTE(enumModbusKodyFunkcji.ZapisBitu),
							uiAdresRejestru := 31 + BYTE_TO_UINT(bKanalEnOcean),
							pZmiennaReferencyjna := 0,
							wWartoscDoZapisania := (BOOL_TO_WORD(FALSE)),
							intModbusOdczytZapisZadanieRozmiar := intModbusOdczytZapisZadanieRozmiar,
							arModbusOdczytZapisZadanie := arModbusOdczytZapisZadanie,
							intModbusOdczytZapisZadanieZnacznikZapisu := intModbusOdczytZapisZadanieZnacznikZapisu);			
END_IF	
//

// Usuwanie siłownika z bramki
IF xUsuwanieHMI THEN	// Usuwanie EnOceanID z bramki
	fnModbusZapisRejestru(	bAdresUrzadzenia := bAdres,																	
							bFunkcja := INT_TO_BYTE(enumModbusKodyFunkcji.ZapisNRejestrow),
							uiAdresRejestru := uintEnOceanIDHiModbusAdres,
							pZmiennaReferencyjna := ADR(wEnOceanIDHi),
							wWartoscDoZapisania := 0,
							intModbusOdczytZapisZadanieRozmiar := intModbusOdczytZapisZadanieRozmiar,
							arModbusOdczytZapisZadanie := arModbusOdczytZapisZadanie,
							intModbusOdczytZapisZadanieZnacznikZapisu := intModbusOdczytZapisZadanieZnacznikZapisu);	
	fnModbusZapisRejestru(	bAdresUrzadzenia := bAdres,																	
							bFunkcja := INT_TO_BYTE(enumModbusKodyFunkcji.ZapisNRejestrow),
							uiAdresRejestru := uintEnOceanIDLoModbusAdres,
							pZmiennaReferencyjna := ADR(wEnOceanIDLo),
							wWartoscDoZapisania := 0,
							intModbusOdczytZapisZadanieRozmiar := intModbusOdczytZapisZadanieRozmiar,
							arModbusOdczytZapisZadanie := arModbusOdczytZapisZadanie,
							intModbusOdczytZapisZadanieZnacznikZapisu := intModbusOdczytZapisZadanieZnacznikZapisu);	
	xUsuwanieHMI := FALSE;					
END_IF
//
(*
// Zmiana koloru - po kliknięciu w symbol siłownika na HMI togglowana jest zmienna xZmienKolorHMI. xResetKoloruHMI resetuje kolor na symbolu, który był kliknięty wcześniej
IF xResetKoloruHMI THEN
	xKolorHMI := FALSE;
	xZmienKolorHMI := FALSE;
END_IF

IF xZmienKolorHMI THEN
	xKolorHMI := TRUE;
END_IF
//
*)
// Detekcja otwarcia okna (jeśli temperatura spadnie w czasie intCzasSpadkuTemperatury o rDeltaSpadkuTemperatury wystaw alarm. Zdejmij alarm, jeśli temp. wzrośnie o rDeltaWzrostuTemperatury
fbDetekcjaOtwarciaOknaTimer(IN := NOT(fbDetekcjaOtwarciaOknaTimer.Q), PT := tCzasSpadkuTemperatury);
IF fbDetekcjaOtwarciaOknaTimer.Q THEN
	rTemperaturaPomieszczeniaHistoryczna := rTemperaturaPomieszczenia;
END_IF
IF (rTemperaturaPomieszczeniaHistoryczna - rTemperaturaPomieszczenia) > rDeltaSpadkuTemperatury THEN
	xAlarmOtwarciaOkna := TRUE;
END_IF
IF (rTemperaturaPomieszczenia - rTemperaturaPomieszczeniaHistoryczna) > rDeltaWzrostuTemperatury THEN
	xAlarmOtwarciaOkna := FALSE;
END_IF
//
// Sprawdzanie czy pomiar temperatury działa (odczyt jest niepoprawny, jeśli nie zmienił wartości w przeciągu doby)
IF rTemperaturaPomieszczeniaPamiec = rTemperaturaPomieszczenia THEN
	xBrakZmianyTemperatury := TRUE;
ELSE
	xBrakZmianyTemperatury := FALSE;	
END_IF
fbBrakZmianyTemperaturyTimer(IN := xBrakZmianyTemperatury, PT := T#12H);
rTemperaturaPomieszczeniaPamiec := rTemperaturaPomieszczenia;
IF fbBrakZmianyTemperaturyTimer.Q AND NOT xBrakKomunikacjiPLC THEN
	xBladBrakZmianyTemperatury := TRUE;
ELSE
	xBladBrakZmianyTemperatury := FALSE;
END_IF
//
///////Diagnostyka na czas uruchomień////////
	rDiagnostykaTemperaturaPomieszczenia := rTemperaturaPomieszczenia;
	rDiagnostykaPozycjaSilownika := rPozycjaSilownika;
	intDiagnostykaFlagaSerwisowa := intFlagaSerwisowa;
	intDiagnostykaTrybPracy := intTrybPracy;
	sDiagnostykaEnOceanIDodczytany := sEnOceanIDodczytany;
	xDiagnostykaPoprawneParowanie := xPoprawneParowanie;
	wDiagnostykaCzasOdOstatniegoKomunikatu := wCzasOdOstatniegoKomunikatu;
//////////////////////////////////////////////				
							
					
//raportowanie		
IF (intBlokadaWykonywaniaRozkazow <> intBlokadaWykonywaniaRozkazowZaraportowana OR intTrybPracy <> intTrybPracyZaraportowana OR rTemperaturaPomieszczenia <> rTemperaturaPomieszczeniaZaraportowana OR 
	rPozycjaSilownika <> rPozycjaSilownikaZaraportowana OR intFlagaSerwisowa <> intFlagaSerwisowaZaraportowana OR rPozycjaSilownikaMan <> rPozycjaSilownikaManZaraportowana OR 
	rPozycjaSilownikaAuto <> rPozycjaSilownikaAutoZaraportowana) AND arModbusStatusKomunikacji[bAdres] = enumModbusStatus.KomunikacjaPrawidlowa AND xPoInicjalizacji THEN
	xRaport := TRUE;
END_IF

IF xRaport THEN
	sDane := '';
	xRaport := FALSE;
	IF intBlokadaWykonywaniaRozkazow <> intBlokadaWykonywaniaRozkazowZaraportowana THEN
		intBlokadaWykonywaniaRozkazowZaraportowana := intBlokadaWykonywaniaRozkazow;
		fnKomunikatDaneDodaj(sDane := sDane , sAtrybut := 'BLOK=' , sWartosc := INT_TO_STRING(intBlokadaWykonywaniaRozkazow));	
	END_IF
	IF intTrybPracy <> intTrybPracyZaraportowana THEN
		intTrybPracyZaraportowana := intTrybPracy;
		fnKomunikatDaneDodaj(sDane := sDane , sAtrybut := 'TRYB=' , sWartosc := INT_TO_STRING(intTrybPracy));	
	END_IF
	IF rTemperaturaPomieszczenia <> rTemperaturaPomieszczeniaZaraportowana THEN
		rTemperaturaPomieszczeniaZaraportowana := rTemperaturaPomieszczenia;
		fnKomunikatDaneDodaj(sDane := sDane , sAtrybut := 'TEMP=' , sWartosc := REAL_TO_STRING(rTemperaturaPomieszczenia));	
	END_IF
	IF rPozycjaSilownika <> rPozycjaSilownikaZaraportowana THEN
		rPozycjaSilownikaZaraportowana := rPozycjaSilownika;
		fnKomunikatDaneDodaj(sDane := sDane , sAtrybut := 'POZ=' , sWartosc := REAL_TO_STRING(rPozycjaSilownika));	
	END_IF
	IF rPozycjaSilownikaMan <> rPozycjaSilownikaManZaraportowana THEN
		rPozycjaSilownikaManZaraportowana := rPozycjaSilownikaMan;
		fnKomunikatDaneDodaj(sDane := sDane , sAtrybut := 'POZMAN=' , sWartosc := REAL_TO_STRING(rPozycjaSilownikaMan / 100));	
	END_IF
	IF rPozycjaSilownikaAuto <> rPozycjaSilownikaAutoZaraportowana THEN
		rPozycjaSilownikaAutoZaraportowana := rPozycjaSilownikaAuto;
		fnKomunikatDaneDodaj(sDane := sDane , sAtrybut := 'POZAUTO=' , sWartosc := REAL_TO_STRING(rPozycjaSilownikaAuto));	
	END_IF
	IF intFlagaSerwisowa <> intFlagaSerwisowaZaraportowana THEN
		intFlagaSerwisowaZaraportowana := intFlagaSerwisowa;
		fnKomunikatDaneDodaj(sDane := sDane , sAtrybut := 'SERWIS=' , sWartosc := INT_TO_STRING(intFlagaSerwisowa));	
	END_IF

	IF sDane <> '' AND xPoInicjalizacji THEN
		fnZapiszKomunikat(	sCalyKomunikat := '' ,
							sTypKomunikatu := 'M' ,
							sMnemonik := sMnemonik ,
							sMACAdres := sMACAdres ,
							sIDNadawcy := sIdInstancji ,
							sIDOdbiorcy := sIdAplikacji ,
							sDaneZapasowe := sDaneZapasowe ,
							sDane := sDane ,
							arTablicaKomunikatow := arTablicaKomunikatow ,
							intTablicaKomunikatowZnacznikZapisu := intTablicaKomunikatowZnacznikZapisu ,
							intTablicaKomunikatowRozmiar := intTablicaKomunikatowRozmiar ,
							sWyslanyKomunikat := sWyslanyKomunikat);
	END_IF
END_IF

// obsługa alarmów do siłownika
	//brak komunikacji po EnOcean
IF arErrorStan[enumPPPSSilownikSABpError.BrakKomunikacji] <> enumAlarmWartosc.StanAlarmowy AND fbTimeoutEnOcean.Q AND arModbusStatusKomunikacji[bAdres] = enumModbusStatus.KomunikacjaPrawidlowa THEN
	arErrorStan[enumPPPSSilownikSABpError.BrakKomunikacji] := enumAlarmWartosc.StanAlarmowy;
	xBrakKomunikacjiEnOcean := TRUE;
	arErrorKlasa[enumPPPSSilownikSABpError.BrakKomunikacji] := enumPPPSSilownikSABpErrorKlasa.BrakKomunikacji;
	IF xPoInicjalizacji THEN
		fnZapiszKomunikat(	sCalyKomunikat := '' ,
							sTypKomunikatu := 'E' ,
							sMnemonik := sMnemonik ,
							sMACAdres := sMACAdres ,
							sIDNadawcy := sIdInstancji ,
							sIDOdbiorcy := sIdAplikacji ,
							sDaneZapasowe := sDaneZapasowe ,
							sDane := fnKomunikatDaneError(xAktywny := TRUE , intKlasa := enumPPPSSilownikSABpErrorKlasa.BrakKomunikacji , intNumer := enumPPPSSilownikSABpError.BrakKomunikacji),
							arTablicaKomunikatow := arTablicaKomunikatow ,
							intTablicaKomunikatowZnacznikZapisu := intTablicaKomunikatowZnacznikZapisu ,
							intTablicaKomunikatowRozmiar := intTablicaKomunikatowRozmiar ,
							sWyslanyKomunikat := sWyslanyKomunikatDummy);
	END_IF
END_IF
IF arErrorStan[enumPPPSSilownikSABpError.BrakKomunikacji] <> enumAlarmWartosc.StanNormalny AND NOT fbTimeoutEnOcean.Q AND arModbusStatusKomunikacji[bAdres] = enumModbusStatus.KomunikacjaPrawidlowa THEN
	arErrorStan[enumPPPSSilownikSABpError.BrakKomunikacji] := enumAlarmWartosc.StanNormalny;
	xBrakKomunikacjiEnOcean := FALSE;
	arErrorKlasa[enumPPPSSilownikSABpError.BrakKomunikacji] := enumPPPSSilownikSABpErrorKlasa.BrakKomunikacji;
	IF xPoInicjalizacji THEN
		fnZapiszKomunikat(	sCalyKomunikat := '' ,
							sTypKomunikatu := 'E' ,
							sMnemonik := sMnemonik ,
							sMACAdres := sMACAdres ,
							sIDNadawcy := sIdInstancji ,
							sIDOdbiorcy := sIdAplikacji ,
							sDaneZapasowe := sDaneZapasowe ,
							sDane := fnKomunikatDaneError(xAktywny := FALSE , intKlasa := enumPPPSSilownikSABpErrorKlasa.BrakKomunikacji , intNumer := enumPPPSSilownikSABpError.BrakKomunikacji),
							arTablicaKomunikatow := arTablicaKomunikatow ,
							intTablicaKomunikatowZnacznikZapisu := intTablicaKomunikatowZnacznikZapisu ,
							intTablicaKomunikatowRozmiar := intTablicaKomunikatowRozmiar ,
							sWyslanyKomunikat := sWyslanyKomunikatDummy);
	END_IF
END_IF
	//Alarm ogólny
IF arErrorStan[enumPPPSSilownikSABpError.AlarmOgolny] <> enumAlarmWartosc.StanAlarmowy AND xAlarmOgolny AND arModbusStatusKomunikacji[bAdres] = enumModbusStatus.KomunikacjaPrawidlowa THEN
	arErrorStan[enumPPPSSilownikSABpError.AlarmOgolny] := enumAlarmWartosc.StanAlarmowy;
	xAwariaUrzadzenia := TRUE;
	arErrorKlasa[enumPPPSSilownikSABpError.AlarmOgolny] := enumPPPSSilownikSABpErrorKlasa.AlarmOgolny;
	IF xPoInicjalizacji THEN
		fnZapiszKomunikat(	sCalyKomunikat := '' ,
							sTypKomunikatu := 'E' ,
							sMnemonik := sMnemonik ,
							sMACAdres := sMACAdres ,
							sIDNadawcy := sIdInstancji ,
							sIDOdbiorcy := sIdAplikacji ,
							sDaneZapasowe := sDaneZapasowe ,
							sDane := fnKomunikatDaneError(xAktywny := TRUE , intKlasa := enumPPPSSilownikSABpErrorKlasa.AlarmOgolny , intNumer := enumPPPSSilownikSABpError.AlarmOgolny),
							arTablicaKomunikatow := arTablicaKomunikatow ,
							intTablicaKomunikatowZnacznikZapisu := intTablicaKomunikatowZnacznikZapisu ,
							intTablicaKomunikatowRozmiar := intTablicaKomunikatowRozmiar ,
							sWyslanyKomunikat := sWyslanyKomunikatDummy);
	END_IF
END_IF
IF arErrorStan[enumPPPSSilownikSABpError.AlarmOgolny] <> enumAlarmWartosc.StanNormalny AND NOT xAlarmOgolny AND arModbusStatusKomunikacji[bAdres] = enumModbusStatus.KomunikacjaPrawidlowa THEN
	arErrorStan[enumPPPSSilownikSABpError.AlarmOgolny] := enumAlarmWartosc.StanNormalny;
	xAwariaUrzadzenia := FALSE;
	arErrorKlasa[enumPPPSSilownikSABpError.AlarmOgolny] := enumPPPSSilownikSABpErrorKlasa.AlarmOgolny;
	IF xPoInicjalizacji THEN
		fnZapiszKomunikat(	sCalyKomunikat := '' ,
							sTypKomunikatu := 'E' ,
							sMnemonik := sMnemonik ,
							sMACAdres := sMACAdres ,
							sIDNadawcy := sIdInstancji ,
							sIDOdbiorcy := sIdAplikacji ,
							sDaneZapasowe := sDaneZapasowe ,
							sDane := fnKomunikatDaneError(xAktywny := FALSE , intKlasa := enumPPPSSilownikSABpErrorKlasa.AlarmOgolny , intNumer := enumPPPSSilownikSABpError.AlarmOgolny),
							arTablicaKomunikatow := arTablicaKomunikatow ,
							intTablicaKomunikatowZnacznikZapisu := intTablicaKomunikatowZnacznikZapisu ,
							intTablicaKomunikatowRozmiar := intTablicaKomunikatowRozmiar ,
							sWyslanyKomunikat := sWyslanyKomunikatDummy);
	END_IF
END_IF
	// Detekcja otwarcia okna
IF arErrorStan[enumPPPSSilownikSABpError.DetekcjaOtwarciaOkna] <> enumAlarmWartosc.StanAlarmowy AND xDetekcjaOtwarciaOkna AND arModbusStatusKomunikacji[bAdres] = enumModbusStatus.KomunikacjaPrawidlowa THEN
	arErrorStan[enumPPPSSilownikSABpError.DetekcjaOtwarciaOkna] := enumAlarmWartosc.StanAlarmowy;
	arErrorKlasa[enumPPPSSilownikSABpError.DetekcjaOtwarciaOkna] := enumPPPSSilownikSABpErrorKlasa.DetekcjaOtwarciaOkna;
	IF xPoInicjalizacji THEN
		fnZapiszKomunikat(	sCalyKomunikat := '' ,
							sTypKomunikatu := 'E' ,
							sMnemonik := sMnemonik ,
							sMACAdres := sMACAdres ,
							sIDNadawcy := sIdInstancji ,
							sIDOdbiorcy := sIdAplikacji ,
							sDaneZapasowe := sDaneZapasowe ,
							sDane := fnKomunikatDaneError(xAktywny := TRUE , intKlasa := enumPPPSSilownikSABpErrorKlasa.DetekcjaOtwarciaOkna , intNumer := enumPPPSSilownikSABpError.DetekcjaOtwarciaOkna),
							arTablicaKomunikatow := arTablicaKomunikatow ,
							intTablicaKomunikatowZnacznikZapisu := intTablicaKomunikatowZnacznikZapisu ,
							intTablicaKomunikatowRozmiar := intTablicaKomunikatowRozmiar ,
							sWyslanyKomunikat := sWyslanyKomunikatDummy);
	END_IF
END_IF
IF arErrorStan[enumPPPSSilownikSABpError.DetekcjaOtwarciaOkna] <> enumAlarmWartosc.StanNormalny AND NOT xDetekcjaOtwarciaOkna AND arModbusStatusKomunikacji[bAdres] = enumModbusStatus.KomunikacjaPrawidlowa THEN
	arErrorStan[enumPPPSSilownikSABpError.DetekcjaOtwarciaOkna] := enumAlarmWartosc.StanNormalny;
	arErrorKlasa[enumPPPSSilownikSABpError.DetekcjaOtwarciaOkna] := enumPPPSSilownikSABpErrorKlasa.DetekcjaOtwarciaOkna;
	IF xPoInicjalizacji THEN
		fnZapiszKomunikat(	sCalyKomunikat := '' ,
							sTypKomunikatu := 'E' ,
							sMnemonik := sMnemonik ,
							sMACAdres := sMACAdres ,
							sIDNadawcy := sIdInstancji ,
							sIDOdbiorcy := sIdAplikacji ,
							sDaneZapasowe := sDaneZapasowe ,
							sDane := fnKomunikatDaneError(xAktywny := FALSE , intKlasa := enumPPPSSilownikSABpErrorKlasa.DetekcjaOtwarciaOkna , intNumer := enumPPPSSilownikSABpError.DetekcjaOtwarciaOkna),
							arTablicaKomunikatow := arTablicaKomunikatow ,
							intTablicaKomunikatowZnacznikZapisu := intTablicaKomunikatowZnacznikZapisu ,
							intTablicaKomunikatowRozmiar := intTablicaKomunikatowRozmiar ,
							sWyslanyKomunikat := sWyslanyKomunikatDummy);
	END_IF
END_IF
// Defrost
IF arErrorStan[enumPPPSSilownikSABpError.Defrost] <> enumAlarmWartosc.StanAlarmowy AND xDefrost AND arModbusStatusKomunikacji[bAdres] = enumModbusStatus.KomunikacjaPrawidlowa THEN
	arErrorStan[enumPPPSSilownikSABpError.Defrost] := enumAlarmWartosc.StanAlarmowy;
	arErrorKlasa[enumPPPSSilownikSABpError.Defrost] := enumPPPSSilownikSABpErrorKlasa.Defrost;
	IF xPoInicjalizacji THEN
		fnZapiszKomunikat(	sCalyKomunikat := '' ,
							sTypKomunikatu := 'E' ,
							sMnemonik := sMnemonik ,
							sMACAdres := sMACAdres ,
							sIDNadawcy := sIdInstancji ,
							sIDOdbiorcy := sIdAplikacji ,
							sDaneZapasowe := sDaneZapasowe ,
							sDane := fnKomunikatDaneError(xAktywny := TRUE , intKlasa := enumPPPSSilownikSABpErrorKlasa.Defrost , intNumer := enumPPPSSilownikSABpError.Defrost),
							arTablicaKomunikatow := arTablicaKomunikatow ,
							intTablicaKomunikatowZnacznikZapisu := intTablicaKomunikatowZnacznikZapisu ,
							intTablicaKomunikatowRozmiar := intTablicaKomunikatowRozmiar ,
							sWyslanyKomunikat := sWyslanyKomunikatDummy);
	END_IF
END_IF
IF arErrorStan[enumPPPSSilownikSABpError.Defrost] <> enumAlarmWartosc.StanNormalny AND NOT xDefrost AND arModbusStatusKomunikacji[bAdres] = enumModbusStatus.KomunikacjaPrawidlowa THEN
	arErrorStan[enumPPPSSilownikSABpError.Defrost] := enumAlarmWartosc.StanNormalny;
	arErrorKlasa[enumPPPSSilownikSABpError.Defrost] := enumPPPSSilownikSABpErrorKlasa.Defrost;
	IF xPoInicjalizacji THEN
		fnZapiszKomunikat(	sCalyKomunikat := '' ,
							sTypKomunikatu := 'E' ,
							sMnemonik := sMnemonik ,
							sMACAdres := sMACAdres ,
							sIDNadawcy := sIdInstancji ,
							sIDOdbiorcy := sIdAplikacji ,
							sDaneZapasowe := sDaneZapasowe ,
							sDane := fnKomunikatDaneError(xAktywny := FALSE , intKlasa := enumPPPSSilownikSABpErrorKlasa.Defrost , intNumer := enumPPPSSilownikSABpError.Defrost),
							arTablicaKomunikatow := arTablicaKomunikatow ,
							intTablicaKomunikatowZnacznikZapisu := intTablicaKomunikatowZnacznikZapisu ,
							intTablicaKomunikatowRozmiar := intTablicaKomunikatowRozmiar ,
							sWyslanyKomunikat := sWyslanyKomunikatDummy);
	END_IF
END_IF
// Alarm czujnika temperatury
IF arErrorStan[enumPPPSSilownikSABpError.AlarmCzujnika] <> enumAlarmWartosc.StanAlarmowy AND xBladBrakZmianyTemperatury AND arModbusStatusKomunikacji[bAdres] = enumModbusStatus.KomunikacjaPrawidlowa THEN
	arErrorStan[enumPPPSSilownikSABpError.AlarmCzujnika] := enumAlarmWartosc.StanAlarmowy;
	arErrorKlasa[enumPPPSSilownikSABpError.AlarmCzujnika] := enumPPPSSilownikSABpErrorKlasa.AlarmCzujnika;
	IF xPoInicjalizacji THEN
		fnZapiszKomunikat(	sCalyKomunikat := '' ,
							sTypKomunikatu := 'E' ,
							sMnemonik := sMnemonik ,
							sMACAdres := sMACAdres ,
							sIDNadawcy := sIdInstancji ,
							sIDOdbiorcy := sIdAplikacji ,
							sDaneZapasowe := sDaneZapasowe ,
							sDane := fnKomunikatDaneError(xAktywny := TRUE , intKlasa := enumPPPSSilownikSABpErrorKlasa.AlarmCzujnika , intNumer := enumPPPSSilownikSABpError.AlarmCzujnika),
							arTablicaKomunikatow := arTablicaKomunikatow ,
							intTablicaKomunikatowZnacznikZapisu := intTablicaKomunikatowZnacznikZapisu ,
							intTablicaKomunikatowRozmiar := intTablicaKomunikatowRozmiar ,
							sWyslanyKomunikat := sWyslanyKomunikatDummy);
	END_IF
END_IF
IF arErrorStan[enumPPPSSilownikSABpError.AlarmCzujnika] <> enumAlarmWartosc.StanNormalny AND NOT xBladBrakZmianyTemperatury AND arModbusStatusKomunikacji[bAdres] = enumModbusStatus.KomunikacjaPrawidlowa THEN
	arErrorStan[enumPPPSSilownikSABpError.AlarmCzujnika] := enumAlarmWartosc.StanNormalny;
	arErrorKlasa[enumPPPSSilownikSABpError.AlarmCzujnika] := enumPPPSSilownikSABpErrorKlasa.AlarmCzujnika;
	IF xPoInicjalizacji THEN
		fnZapiszKomunikat(	sCalyKomunikat := '' ,
							sTypKomunikatu := 'E' ,
							sMnemonik := sMnemonik ,
							sMACAdres := sMACAdres ,
							sIDNadawcy := sIdInstancji ,
							sIDOdbiorcy := sIdAplikacji ,
							sDaneZapasowe := sDaneZapasowe ,
							sDane := fnKomunikatDaneError(xAktywny := FALSE , intKlasa := enumPPPSSilownikSABpErrorKlasa.AlarmCzujnika , intNumer := enumPPPSSilownikSABpError.AlarmCzujnika),
							arTablicaKomunikatow := arTablicaKomunikatow ,
							intTablicaKomunikatowZnacznikZapisu := intTablicaKomunikatowZnacznikZapisu ,
							intTablicaKomunikatowRozmiar := intTablicaKomunikatowRozmiar ,
							sWyslanyKomunikat := sWyslanyKomunikatDummy);
	END_IF
END_IF

          
END_FUNCTION_BLOCK
